(* IEC 61131-3 sources: myCodes/Stone/Rohit-AddOnsTesting/Rohit-AddOnsTesting/Generated, 4 files *)

(* ---- System.Globalization.g.st ---- *)
//********************************************************************//
//*               System.globalization generated file                *//
//********************************************************************//

NAMESPACE System.Globalization

TYPE { ATTRIBUTE ENUM_SIZE 2 } UOM :
(
	NONE,
	YEAR,
	WEEK,
	DAY,
	HOUR,
	MINUTE,
	MONTH,
	SECOND,
	HUNDREDTHS_SECOND,
	MILLISECOND,
	MICROSECOND,
	MICROMETER,
	MILLIMETER,
	CENTIMETER,
	METER,
	KILOMETER,
	INCH,
	FOOT,
	MILE,
	YARD,
	MILLIGRAM,
	GRAM,
	KILOGRAM,
	OUNCE,
	POUND,
	TON,
	TON_REFRIGERATION,
	POUND_MASS,
	POUND_FORCE,
	SQUARE_METER,
	SQUARE_KILOMETER,
	SQUARE_FOOT,
	SQUARE_INCH,
	SQUARE_MILE,
	SQUARE_YARD,
	HECTARE,
	ACRE,
	MILLILITER,
	CENTILITER,
	LITER,
	CUBIC_METER,
	CUBIC_FOOT,
	CUBIC_INCH,
	IMPERIAL_GALLON,
	US_GALLON,
	CELSIUS,
	TENTHS_CELSIUS,
	FAHRENHEIT,
	KELVIN,
	DELTAKELVIN,
	DELTAFAHRENHEIT,
	CELSIUS_PER_HOUR,
	CELSIUS_PER_MINUTE,
	FAHRENHEIT_PER_HOUR,
	FAHRENHEIT_PER_MINUTE,
	ATMOSPHERE,
	BAR,
	TENTHS_BAR,
	MILLIBAR,
	PSI,
	PASCAL,
	HECTOPASCAL,
	KILOPASCAL,
	WATER_CENTIMETER,
	WATER_INCH,
	MERCURY_MILLIMETER,
	MERCURY_CENTIMETER,
	MERCURY_INCH,
	PRESSURE_PASCAL,
	PRESSURE_WATER_INCH,
	PERCENT,
	TENTHS_PERCENT,
	MILLIOHM,
	OHM,
	KILOOHM,
	MEGAOHM,
	MILLIVOLT,
	VOLT,
	MEGAVOLT,
	MILLIAMPERE,
	AMPERE,
	VOLT_AMPERE,
	KILOVOLT_AMPERE,
	MEGAVOLT_AMPERE,
	MICROSIEMENS,
	MILLISIEMENS,
	SIEMENS,
	VOLT_AMPERE_REACTIVE,
	KILOVOLT_AMPERE_REACTIVE,
	MEGAVOLT_AMPERE_REACTIVE,
	NEWTON,
	NEWTON_METER,
	POUND_FOOT,
	POUND_PER_SQUARE_INCH,
	POUND_FORCE_PER_SQUARE_INCH,
	MILLIWATT,
	WATT,
	KILOWATT,
	MEGAWATT,
	WATT_HOUR,
	KILOWATT_HOUR,
	MEGAWATT_HOUR,
	WATT_PER_SQUARE_METER,
	WATT_PER_SQUARE_FOOT,
	HORSEPOWER,
	THERMAL_POWER_BTU,
	THERMAL_POWER_BTU_PER_HOUR,
	REFRIGERATION_POWER_KILOWATT,
	THERMAL_POWER_WATT,
	ELECTRICAL_POWER_WATT,
	JOULE,
	KILOJOULE,
	MEGAJOULE,
	JOULE_PER_KELVIN,
	KILOJOULE_PER_KELVIN,
	MEGAJOULE_PER_KELVIN,
	JOULE_PER_KILOGRAM_KELVIN,
	JOULE_SECOND,
	JOULE_PER_SECOND,
	JOULE_PER_GRAM,
	JOULE_PER_KILOGRAM,
	KILOJOULE_PER_KILOGRAM,
	MEGAJOULE_PER_KILOGRAM,
	BTU,
	KILOBTU,
	MEGABTU,
	KILOBTU_PER_HOUR,
	BTU_PER_POUND,
	BTU_PER_HOUR,
	CALORIE,
	KILOCALORIE_PER_KILOGRAM,
	LUMEN,
	LUX,
	FOOT_CANDLE,
	CANDELA,
	CANDELA_PER_SQUARE_METER,
	GRAM_KELVIN,
	KILOGRAM_KELVIN,
	ENTALPHY_KILOJOULE,
	ENTALPHY_BTU,
	DRY_AIR_KILOGRAM,
	DRY_AIR_POUND,
	KILOJOULE_PER_DRY_AIR_KILOGRAM,
	MEGAJOULE_PER_DRY_AIR_KILOGRAM,
	ENTALPHY_KILOJOULE_PER_KILOGRAM,
	ENTALPHY_BTU_PER_POUND,
	JOULE_PER_DRY_AIR_KILOGRAM,
	BTU_PER_DRY_AIR_POUND,
	METER_PER_SECOND,
	METER_PER_MINUTE,
	KILOMETER_PER_HOUR,
	FOOT_PER_SECOND,
	FOOT_PER_MINUTE,
	MILE_PER_HOUR,
	RPS,
	RPM,
	HERTZ,
	KILOHERTZ,
	MEGAHERTZ,
	CUBIC_METER_PER_SECOND,
	CUBIC_METER_PER_MINUTE,
	CUBIC_METER_PER_HOUR,
	CUBIC_FOOT_PER_HOUR,
	CUBIC_FOOT_PER_MINUTE,
	CUBIC_FOOT_PER_SECOND,
	IMPERIAL_GALLON_PER_SECOND,
	IMPERIAL_GALLON_PER_MINUTE,
	US_GALLON_PER_SECOND,
	US_GALLON_PER_MINUTE,
	US_GALLON_PER_HOUR,
	LITER_PER_SECOND,
	LITER_PER_MINUTE,
	LITER_PER_HOUR,
	TON_HOUR,
	TON_PER_HOUR,
	GRAM_PER_SECOND,
	GRAM_PER_MINUTE,
	GRAM_PER_HOUR,
	KILOGRAM_PER_SECOND,
	KILOGRAM_PER_MINUTE,
	KILOGRAM_PER_HOUR,
	POUND_PER_MINUTE,
	POUND_PER_HOUR,
	GRAM_PER_KILOGRAM,
	TENTHS_GRAM_PER_KILOGRAM,
	KILOGRAM_PER_CUBIC_METER,
	AIR_FLOW_CUBIC_METER,
	AIR_FLOW_CUBIC_FOOT,
	AIR_FLOW_CUBIC_METER_PER_HOUR,
	AIR_FLOW_CUBIC_FOOT_PER_MINUTE,
	WATER_KILOGRAM_PER_DRY_AIR_KILOGRAM,
	TENTHS_WATER_KILOGRAM_PER_DRY_AIR_KILOGRAM,
	PERCENT_rH,
	TENTHS_PERCENT_rH,
	WATER_KILOGRAM,
	WATER_GRAM,
	WATER_GRAM_PER_DRY_AIR_KILOGRAM,
	TENTHS_WATER_GRAM_PER_DRY_AIR_KILOGRAM,
	DELTACELSIUS,
	HENRY,
	MILLIHENRY,
	PPM,
	PPB,
	HERTZ_PER_SECOND,
	CYCLE_PER_SECOND,
	STEPS
);
END_TYPE

{ATTRIBUTE NATIVE}
FUNCTION UOM_OF : UOM
	VAR_INPUT IN : ANY_NUM; END_VAR
END_FUNCTION

TYPE UOM_REAL:
UNION
	VALUE : REAL;
	{ATTRIBUTE UOM YEAR}
	YEAR : REAL;
	{ATTRIBUTE UOM WEEK}
	WEEK : REAL;
	{ATTRIBUTE UOM DAY}
	DAY : REAL;
	{ATTRIBUTE UOM HOUR}
	HOUR : REAL;
	{ATTRIBUTE UOM MINUTE}
	MINUTE : REAL;
	{ATTRIBUTE UOM MONTH}
	MONTH : REAL;
	{ATTRIBUTE UOM SECOND}
	SECOND : REAL;
	{ATTRIBUTE UOM HUNDREDTHS_SECOND}
	HUNDREDTHS_SECOND : REAL;
	{ATTRIBUTE UOM MILLISECOND}
	MILLISECOND : REAL;
	{ATTRIBUTE UOM MICROSECOND}
	MICROSECOND : REAL;
	{ATTRIBUTE UOM MICROMETER}
	MICROMETER : REAL;
	{ATTRIBUTE UOM MILLIMETER}
	MILLIMETER : REAL;
	{ATTRIBUTE UOM CENTIMETER}
	CENTIMETER : REAL;
	{ATTRIBUTE UOM METER}
	METER : REAL;
	{ATTRIBUTE UOM KILOMETER}
	KILOMETER : REAL;
	{ATTRIBUTE UOM INCH}
	INCH : REAL;
	{ATTRIBUTE UOM FOOT}
	FOOT : REAL;
	{ATTRIBUTE UOM MILE}
	MILE : REAL;
	{ATTRIBUTE UOM YARD}
	YARD : REAL;
	{ATTRIBUTE UOM MILLIGRAM}
	MILLIGRAM : REAL;
	{ATTRIBUTE UOM GRAM}
	GRAM : REAL;
	{ATTRIBUTE UOM KILOGRAM}
	KILOGRAM : REAL;
	{ATTRIBUTE UOM OUNCE}
	OUNCE : REAL;
	{ATTRIBUTE UOM POUND}
	POUND : REAL;
	{ATTRIBUTE UOM TON}
	TON : REAL;
	{ATTRIBUTE UOM TON_REFRIGERATION}
	TON_REFRIGERATION : REAL;
	{ATTRIBUTE UOM POUND_MASS}
	POUND_MASS : REAL;
	{ATTRIBUTE UOM POUND_FORCE}
	POUND_FORCE : REAL;
	{ATTRIBUTE UOM SQUARE_METER}
	SQUARE_METER : REAL;
	{ATTRIBUTE UOM SQUARE_KILOMETER}
	SQUARE_KILOMETER : REAL;
	{ATTRIBUTE UOM SQUARE_FOOT}
	SQUARE_FOOT : REAL;
	{ATTRIBUTE UOM SQUARE_INCH}
	SQUARE_INCH : REAL;
	{ATTRIBUTE UOM SQUARE_MILE}
	SQUARE_MILE : REAL;
	{ATTRIBUTE UOM SQUARE_YARD}
	SQUARE_YARD : REAL;
	{ATTRIBUTE UOM HECTARE}
	HECTARE : REAL;
	{ATTRIBUTE UOM ACRE}
	ACRE : REAL;
	{ATTRIBUTE UOM MILLILITER}
	MILLILITER : REAL;
	{ATTRIBUTE UOM CENTILITER}
	CENTILITER : REAL;
	{ATTRIBUTE UOM LITER}
	LITER : REAL;
	{ATTRIBUTE UOM CUBIC_METER}
	CUBIC_METER : REAL;
	{ATTRIBUTE UOM CUBIC_FOOT}
	CUBIC_FOOT : REAL;
	{ATTRIBUTE UOM CUBIC_INCH}
	CUBIC_INCH : REAL;
	{ATTRIBUTE UOM IMPERIAL_GALLON}
	IMPERIAL_GALLON : REAL;
	{ATTRIBUTE UOM US_GALLON}
	US_GALLON : REAL;
	{ATTRIBUTE UOM CELSIUS}
	CELSIUS : REAL;
	{ATTRIBUTE UOM TENTHS_CELSIUS}
	TENTHS_CELSIUS : REAL;
	{ATTRIBUTE UOM FAHRENHEIT}
	FAHRENHEIT : REAL;
	{ATTRIBUTE UOM KELVIN}
	KELVIN : REAL;
	{ATTRIBUTE UOM DELTAKELVIN}
	DELTAKELVIN : REAL;
	{ATTRIBUTE UOM DELTAFAHRENHEIT}
	DELTAFAHRENHEIT : REAL;
	{ATTRIBUTE UOM CELSIUS_PER_HOUR}
	CELSIUS_PER_HOUR : REAL;
	{ATTRIBUTE UOM CELSIUS_PER_MINUTE}
	CELSIUS_PER_MINUTE : REAL;
	{ATTRIBUTE UOM FAHRENHEIT_PER_HOUR}
	FAHRENHEIT_PER_HOUR : REAL;
	{ATTRIBUTE UOM FAHRENHEIT_PER_MINUTE}
	FAHRENHEIT_PER_MINUTE : REAL;
	{ATTRIBUTE UOM ATMOSPHERE}
	ATMOSPHERE : REAL;
	{ATTRIBUTE UOM BAR}
	BAR : REAL;
	{ATTRIBUTE UOM TENTHS_BAR}
	TENTHS_BAR : REAL;
	{ATTRIBUTE UOM MILLIBAR}
	MILLIBAR : REAL;
	{ATTRIBUTE UOM PSI}
	PSI : REAL;
	{ATTRIBUTE UOM PASCAL}
	PASCAL : REAL;
	{ATTRIBUTE UOM HECTOPASCAL}
	HECTOPASCAL : REAL;
	{ATTRIBUTE UOM KILOPASCAL}
	KILOPASCAL : REAL;
	{ATTRIBUTE UOM WATER_CENTIMETER}
	WATER_CENTIMETER : REAL;
	{ATTRIBUTE UOM WATER_INCH}
	WATER_INCH : REAL;
	{ATTRIBUTE UOM MERCURY_MILLIMETER}
	MERCURY_MILLIMETER : REAL;
	{ATTRIBUTE UOM MERCURY_CENTIMETER}
	MERCURY_CENTIMETER : REAL;
	{ATTRIBUTE UOM MERCURY_INCH}
	MERCURY_INCH : REAL;
	{ATTRIBUTE UOM PRESSURE_PASCAL}
	PRESSURE_PASCAL : REAL;
	{ATTRIBUTE UOM PRESSURE_WATER_INCH}
	PRESSURE_WATER_INCH : REAL;
	{ATTRIBUTE UOM PERCENT}
	PERCENT : REAL;
	{ATTRIBUTE UOM TENTHS_PERCENT}
	TENTHS_PERCENT : REAL;
	{ATTRIBUTE UOM MILLIOHM}
	MILLIOHM : REAL;
	{ATTRIBUTE UOM OHM}
	OHM : REAL;
	{ATTRIBUTE UOM KILOOHM}
	KILOOHM : REAL;
	{ATTRIBUTE UOM MEGAOHM}
	MEGAOHM : REAL;
	{ATTRIBUTE UOM MILLIVOLT}
	MILLIVOLT : REAL;
	{ATTRIBUTE UOM VOLT}
	VOLT : REAL;
	{ATTRIBUTE UOM MEGAVOLT}
	MEGAVOLT : REAL;
	{ATTRIBUTE UOM MILLIAMPERE}
	MILLIAMPERE : REAL;
	{ATTRIBUTE UOM AMPERE}
	AMPERE : REAL;
	{ATTRIBUTE UOM VOLT_AMPERE}
	VOLT_AMPERE : REAL;
	{ATTRIBUTE UOM KILOVOLT_AMPERE}
	KILOVOLT_AMPERE : REAL;
	{ATTRIBUTE UOM MEGAVOLT_AMPERE}
	MEGAVOLT_AMPERE : REAL;
	{ATTRIBUTE UOM MICROSIEMENS}
	MICROSIEMENS : REAL;
	{ATTRIBUTE UOM MILLISIEMENS}
	MILLISIEMENS : REAL;
	{ATTRIBUTE UOM SIEMENS}
	SIEMENS : REAL;
	{ATTRIBUTE UOM VOLT_AMPERE_REACTIVE}
	VOLT_AMPERE_REACTIVE : REAL;
	{ATTRIBUTE UOM KILOVOLT_AMPERE_REACTIVE}
	KILOVOLT_AMPERE_REACTIVE : REAL;
	{ATTRIBUTE UOM MEGAVOLT_AMPERE_REACTIVE}
	MEGAVOLT_AMPERE_REACTIVE : REAL;
	{ATTRIBUTE UOM NEWTON}
	NEWTON : REAL;
	{ATTRIBUTE UOM NEWTON_METER}
	NEWTON_METER : REAL;
	{ATTRIBUTE UOM POUND_FOOT}
	POUND_FOOT : REAL;
	{ATTRIBUTE UOM POUND_PER_SQUARE_INCH}
	POUND_PER_SQUARE_INCH : REAL;
	{ATTRIBUTE UOM POUND_FORCE_PER_SQUARE_INCH}
	POUND_FORCE_PER_SQUARE_INCH : REAL;
	{ATTRIBUTE UOM MILLIWATT}
	MILLIWATT : REAL;
	{ATTRIBUTE UOM WATT}
	WATT : REAL;
	{ATTRIBUTE UOM KILOWATT}
	KILOWATT : REAL;
	{ATTRIBUTE UOM MEGAWATT}
	MEGAWATT : REAL;
	{ATTRIBUTE UOM WATT_HOUR}
	WATT_HOUR : REAL;
	{ATTRIBUTE UOM KILOWATT_HOUR}
	KILOWATT_HOUR : REAL;
	{ATTRIBUTE UOM MEGAWATT_HOUR}
	MEGAWATT_HOUR : REAL;
	{ATTRIBUTE UOM WATT_PER_SQUARE_METER}
	WATT_PER_SQUARE_METER : REAL;
	{ATTRIBUTE UOM WATT_PER_SQUARE_FOOT}
	WATT_PER_SQUARE_FOOT : REAL;
	{ATTRIBUTE UOM HORSEPOWER}
	HORSEPOWER : REAL;
	{ATTRIBUTE UOM THERMAL_POWER_BTU}
	THERMAL_POWER_BTU : REAL;
	{ATTRIBUTE UOM THERMAL_POWER_BTU_PER_HOUR}
	THERMAL_POWER_BTU_PER_HOUR : REAL;
	{ATTRIBUTE UOM REFRIGERATION_POWER_KILOWATT}
	REFRIGERATION_POWER_KILOWATT : REAL;
	{ATTRIBUTE UOM THERMAL_POWER_WATT}
	THERMAL_POWER_WATT : REAL;
	{ATTRIBUTE UOM ELECTRICAL_POWER_WATT}
	ELECTRICAL_POWER_WATT : REAL;
	{ATTRIBUTE UOM JOULE}
	JOULE : REAL;
	{ATTRIBUTE UOM KILOJOULE}
	KILOJOULE : REAL;
	{ATTRIBUTE UOM MEGAJOULE}
	MEGAJOULE : REAL;
	{ATTRIBUTE UOM JOULE_PER_KELVIN}
	JOULE_PER_KELVIN : REAL;
	{ATTRIBUTE UOM KILOJOULE_PER_KELVIN}
	KILOJOULE_PER_KELVIN : REAL;
	{ATTRIBUTE UOM MEGAJOULE_PER_KELVIN}
	MEGAJOULE_PER_KELVIN : REAL;
	{ATTRIBUTE UOM JOULE_PER_KILOGRAM_KELVIN}
	JOULE_PER_KILOGRAM_KELVIN : REAL;
	{ATTRIBUTE UOM JOULE_SECOND}
	JOULE_SECOND : REAL;
	{ATTRIBUTE UOM JOULE_PER_SECOND}
	JOULE_PER_SECOND : REAL;
	{ATTRIBUTE UOM JOULE_PER_GRAM}
	JOULE_PER_GRAM : REAL;
	{ATTRIBUTE UOM JOULE_PER_KILOGRAM}
	JOULE_PER_KILOGRAM : REAL;
	{ATTRIBUTE UOM KILOJOULE_PER_KILOGRAM}
	KILOJOULE_PER_KILOGRAM : REAL;
	{ATTRIBUTE UOM MEGAJOULE_PER_KILOGRAM}
	MEGAJOULE_PER_KILOGRAM : REAL;
	{ATTRIBUTE UOM BTU}
	BTU : REAL;
	{ATTRIBUTE UOM KILOBTU}
	KILOBTU : REAL;
	{ATTRIBUTE UOM MEGABTU}
	MEGABTU : REAL;
	{ATTRIBUTE UOM KILOBTU_PER_HOUR}
	KILOBTU_PER_HOUR : REAL;
	{ATTRIBUTE UOM BTU_PER_POUND}
	BTU_PER_POUND : REAL;
	{ATTRIBUTE UOM BTU_PER_HOUR}
	BTU_PER_HOUR : REAL;
	{ATTRIBUTE UOM CALORIE}
	CALORIE : REAL;
	{ATTRIBUTE UOM KILOCALORIE_PER_KILOGRAM}
	KILOCALORIE_PER_KILOGRAM : REAL;
	{ATTRIBUTE UOM LUMEN}
	LUMEN : REAL;
	{ATTRIBUTE UOM LUX}
	LUX : REAL;
	{ATTRIBUTE UOM FOOT_CANDLE}
	FOOT_CANDLE : REAL;
	{ATTRIBUTE UOM CANDELA}
	CANDELA : REAL;
	{ATTRIBUTE UOM CANDELA_PER_SQUARE_METER}
	CANDELA_PER_SQUARE_METER : REAL;
	{ATTRIBUTE UOM GRAM_KELVIN}
	GRAM_KELVIN : REAL;
	{ATTRIBUTE UOM KILOGRAM_KELVIN}
	KILOGRAM_KELVIN : REAL;
	{ATTRIBUTE UOM ENTALPHY_KILOJOULE}
	ENTALPHY_KILOJOULE : REAL;
	{ATTRIBUTE UOM ENTALPHY_BTU}
	ENTALPHY_BTU : REAL;
	{ATTRIBUTE UOM DRY_AIR_KILOGRAM}
	DRY_AIR_KILOGRAM : REAL;
	{ATTRIBUTE UOM DRY_AIR_POUND}
	DRY_AIR_POUND : REAL;
	{ATTRIBUTE UOM KILOJOULE_PER_DRY_AIR_KILOGRAM}
	KILOJOULE_PER_DRY_AIR_KILOGRAM : REAL;
	{ATTRIBUTE UOM MEGAJOULE_PER_DRY_AIR_KILOGRAM}
	MEGAJOULE_PER_DRY_AIR_KILOGRAM : REAL;
	{ATTRIBUTE UOM ENTALPHY_KILOJOULE_PER_KILOGRAM}
	ENTALPHY_KILOJOULE_PER_KILOGRAM : REAL;
	{ATTRIBUTE UOM ENTALPHY_BTU_PER_POUND}
	ENTALPHY_BTU_PER_POUND : REAL;
	{ATTRIBUTE UOM JOULE_PER_DRY_AIR_KILOGRAM}
	JOULE_PER_DRY_AIR_KILOGRAM : REAL;
	{ATTRIBUTE UOM BTU_PER_DRY_AIR_POUND}
	BTU_PER_DRY_AIR_POUND : REAL;
	{ATTRIBUTE UOM METER_PER_SECOND}
	METER_PER_SECOND : REAL;
	{ATTRIBUTE UOM METER_PER_MINUTE}
	METER_PER_MINUTE : REAL;
	{ATTRIBUTE UOM KILOMETER_PER_HOUR}
	KILOMETER_PER_HOUR : REAL;
	{ATTRIBUTE UOM FOOT_PER_SECOND}
	FOOT_PER_SECOND : REAL;
	{ATTRIBUTE UOM FOOT_PER_MINUTE}
	FOOT_PER_MINUTE : REAL;
	{ATTRIBUTE UOM MILE_PER_HOUR}
	MILE_PER_HOUR : REAL;
	{ATTRIBUTE UOM RPS}
	RPS : REAL;
	{ATTRIBUTE UOM RPM}
	RPM : REAL;
	{ATTRIBUTE UOM HERTZ}
	HERTZ : REAL;
	{ATTRIBUTE UOM KILOHERTZ}
	KILOHERTZ : REAL;
	{ATTRIBUTE UOM MEGAHERTZ}
	MEGAHERTZ : REAL;
	{ATTRIBUTE UOM CUBIC_METER_PER_SECOND}
	CUBIC_METER_PER_SECOND : REAL;
	{ATTRIBUTE UOM CUBIC_METER_PER_MINUTE}
	CUBIC_METER_PER_MINUTE : REAL;
	{ATTRIBUTE UOM CUBIC_METER_PER_HOUR}
	CUBIC_METER_PER_HOUR : REAL;
	{ATTRIBUTE UOM CUBIC_FOOT_PER_HOUR}
	CUBIC_FOOT_PER_HOUR : REAL;
	{ATTRIBUTE UOM CUBIC_FOOT_PER_MINUTE}
	CUBIC_FOOT_PER_MINUTE : REAL;
	{ATTRIBUTE UOM CUBIC_FOOT_PER_SECOND}
	CUBIC_FOOT_PER_SECOND : REAL;
	{ATTRIBUTE UOM IMPERIAL_GALLON_PER_SECOND}
	IMPERIAL_GALLON_PER_SECOND : REAL;
	{ATTRIBUTE UOM IMPERIAL_GALLON_PER_MINUTE}
	IMPERIAL_GALLON_PER_MINUTE : REAL;
	{ATTRIBUTE UOM US_GALLON_PER_SECOND}
	US_GALLON_PER_SECOND : REAL;
	{ATTRIBUTE UOM US_GALLON_PER_MINUTE}
	US_GALLON_PER_MINUTE : REAL;
	{ATTRIBUTE UOM US_GALLON_PER_HOUR}
	US_GALLON_PER_HOUR : REAL;
	{ATTRIBUTE UOM LITER_PER_SECOND}
	LITER_PER_SECOND : REAL;
	{ATTRIBUTE UOM LITER_PER_MINUTE}
	LITER_PER_MINUTE : REAL;
	{ATTRIBUTE UOM LITER_PER_HOUR}
	LITER_PER_HOUR : REAL;
	{ATTRIBUTE UOM TON_HOUR}
	TON_HOUR : REAL;
	{ATTRIBUTE UOM TON_PER_HOUR}
	TON_PER_HOUR : REAL;
	{ATTRIBUTE UOM GRAM_PER_SECOND}
	GRAM_PER_SECOND : REAL;
	{ATTRIBUTE UOM GRAM_PER_MINUTE}
	GRAM_PER_MINUTE : REAL;
	{ATTRIBUTE UOM GRAM_PER_HOUR}
	GRAM_PER_HOUR : REAL;
	{ATTRIBUTE UOM KILOGRAM_PER_SECOND}
	KILOGRAM_PER_SECOND : REAL;
	{ATTRIBUTE UOM KILOGRAM_PER_MINUTE}
	KILOGRAM_PER_MINUTE : REAL;
	{ATTRIBUTE UOM KILOGRAM_PER_HOUR}
	KILOGRAM_PER_HOUR : REAL;
	{ATTRIBUTE UOM POUND_PER_MINUTE}
	POUND_PER_MINUTE : REAL;
	{ATTRIBUTE UOM POUND_PER_HOUR}
	POUND_PER_HOUR : REAL;
	{ATTRIBUTE UOM GRAM_PER_KILOGRAM}
	GRAM_PER_KILOGRAM : REAL;
	{ATTRIBUTE UOM TENTHS_GRAM_PER_KILOGRAM}
	TENTHS_GRAM_PER_KILOGRAM : REAL;
	{ATTRIBUTE UOM KILOGRAM_PER_CUBIC_METER}
	KILOGRAM_PER_CUBIC_METER : REAL;
	{ATTRIBUTE UOM AIR_FLOW_CUBIC_METER}
	AIR_FLOW_CUBIC_METER : REAL;
	{ATTRIBUTE UOM AIR_FLOW_CUBIC_FOOT}
	AIR_FLOW_CUBIC_FOOT : REAL;
	{ATTRIBUTE UOM AIR_FLOW_CUBIC_METER_PER_HOUR}
	AIR_FLOW_CUBIC_METER_PER_HOUR : REAL;
	{ATTRIBUTE UOM AIR_FLOW_CUBIC_FOOT_PER_MINUTE}
	AIR_FLOW_CUBIC_FOOT_PER_MINUTE : REAL;
	{ATTRIBUTE UOM WATER_KILOGRAM_PER_DRY_AIR_KILOGRAM}
	WATER_KILOGRAM_PER_DRY_AIR_KILOGRAM : REAL;
	{ATTRIBUTE UOM TENTHS_WATER_KILOGRAM_PER_DRY_AIR_KILOGRAM}
	TENTHS_WATER_KILOGRAM_PER_DRY_AIR_KILOGRAM : REAL;
	{ATTRIBUTE UOM PERCENT_rH}
	PERCENT_rH : REAL;
	{ATTRIBUTE UOM TENTHS_PERCENT_rH}
	TENTHS_PERCENT_rH : REAL;
	{ATTRIBUTE UOM WATER_KILOGRAM}
	WATER_KILOGRAM : REAL;
	{ATTRIBUTE UOM WATER_GRAM}
	WATER_GRAM : REAL;
	{ATTRIBUTE UOM WATER_GRAM_PER_DRY_AIR_KILOGRAM}
	WATER_GRAM_PER_DRY_AIR_KILOGRAM : REAL;
	{ATTRIBUTE UOM TENTHS_WATER_GRAM_PER_DRY_AIR_KILOGRAM}
	TENTHS_WATER_GRAM_PER_DRY_AIR_KILOGRAM : REAL;
	{ATTRIBUTE UOM DELTACELSIUS}
	DELTACELSIUS : REAL;
	{ATTRIBUTE UOM HENRY}
	HENRY : REAL;
	{ATTRIBUTE UOM MILLIHENRY}
	MILLIHENRY : REAL;
	{ATTRIBUTE UOM PPM}
	PPM : REAL;
	{ATTRIBUTE UOM PPB}
	PPB : REAL;
	{ATTRIBUTE UOM HERTZ_PER_SECOND}
	HERTZ_PER_SECOND : REAL;
	{ATTRIBUTE UOM CYCLE_PER_SECOND}
	CYCLE_PER_SECOND : REAL;
	{ATTRIBUTE UOM STEPS}
	STEPS : REAL;
END_UNION;
END_TYPE
END_NAMESPACE

(* ---- Assets.g.st ---- *)
//********************************************************************//
//*                      Assets generated file                       *//
//********************************************************************//

NAMESPACE Assets.Language

VAR_GLOBAL CONSTANT
	_EN: UINT := 1;

	ResMap : ARRAY[1..1] OF STRING :=
	[
		'EN'
	];
END_VAR

END_NAMESPACE

(* ---- Assets.Strings.g.st ---- *)
NAMESPACE Assets.Language

VAR_GLOBAL CONSTANT
	LanguagesCount : UINT := 1;
END_VAR

END_NAMESPACE

(* ---- System.IO.g.st ---- *)
//********************************************************************//
//*                   System.IO generated file                       *//
//********************************************************************//

NAMESPACE System.IO

VAR_GLOBAL CONSTANT
	(** Max number of universal channels *)
	LIB_IO_MAX_U_CH : USINT := 11;
	(** Max number of analog channels *)
	LIB_IO_MAX_Y_CH : USINT := 4;
	(** Max number of NO channels *)
	LIB_IO_MAX_NO_CH : USINT := 6;
	(** Max number of ID channels *)
	LIB_IO_MAX_ID_CH : USINT := 8;
END_VAR

END_NAMESPACE
